Fanuc KAREL source: ko00045.KL

-- PROVISIONAL review KL for V770-1; original PC SHA256 f8390df0685be9174fb15b59b63358aeb7d727a48757fbacac7bea9918f48c65
-- Incomplete behavior may be omitted. Consult companion uncertainty JSON. Do not deploy.
PROGRAM KO00045
%NOLOCKGROUP
BEGIN
  -- UNRESOLVED_PC offsets 5-12; opcodes 9D,23
  -- UNRESOLVED_PC offsets 17-69; opcodes 27,27,49,7E,AD,27,49,7E,AD,22,31,7E,4A
  -- UNRESOLVED_PC offsets 74-78; opcodes 7F
END KO00045
